FUNCTION_BLOCK FB_Keypad_4x2_Tap
VAR_INPUT
	Key: ARRAY [0..7] OF ST_DigitalInput;
END_VAR
VAR_OUTPUT
	KeyEvent: ARRAY[0..7] OF BOOL;
END_VAR
VAR
	
END_VAR

END_FUNCTION_BLOCK

(* stored: Version 1.1.0.1, ProductVersion 3.1.4024.12
   POU FB_Keypad_4x2_Tap: Id {62204366-1607-4ea6-aa09-a6fea29f7c55}, SpecialFunc None *)
